PROGRAM pActvOutputs

(*Activar Salidas BOMBA CIRCULACION*)
Z_CP();

(*Activar Salidas control*)
z_control();

(*Activar Salidas drain*)
z_drain();

(*Activar Salidas fILL*)
z_FILL();

(*Activar Salidas LEVEL*)
z_level();

(*Activar Salidas pRESS*)
z_press();

(*Activar Salidas tk1*)
z_TK1();

(*Activar Salidas tk2*)
z_TK2();

(*Activar Salidas CIRC*)
Z_CIRC();

(*Activar Salidas TERMo*)
Z_TEMP();

(*Activar Salidas OVERFLOW*)
z_OVERFLOW();

(*Activar Salidas INTRO*)
z_INTRO();

END_PROGRAM

(* stored: Version 1.1.0.1, ProductVersion 3.1.4024.10
   POU pActvOutputs: Id {7c4f79d2-73ba-4371-a326-61c07187c10b}, SpecialFunc None *)
